// TIA Portal project "Siemens_B3" (V16)

(* hardware
DEVICE "S7-1200 station_1"  S7-1200 Station
   slot 0: "Rack_0"  S7-1200 Rack  Rack  V1.0
   slot 1: "PLC_1"  CPU 1214C DC/DC/DC  6ES7 214-1AG40-0XB0  V4.0
   slot 3: "AQ 1x12BIT_1"  AQ1 signal board  6ES7 232-4HA30-0XB0  V1.0
DEVICE "PC-System_2"  SIMATIC PC station
   slot 0: "SIMATIC PC station"  Rail  SIMATIC PC-Station  V1.0
      slot 125: "Stationmanager"  Station_Manager  V6.0.4
   slot 1: "HMI_RT_2"  WinCC RT Professional  6AV2 105-0xxxx-xxxx  16.0.0.0
   slot 2: "IE general_1"  IE General  IE_CP  V8.2.0
DEVICE "PC-System_1"  SIMATIC PC station
   slot 0: "SIMATIC PC station"  Rail  SIMATIC PC-Station  V1.0
      slot 125: "Stationmanager"  Station_Manager  V6.0.4
   slot 1: "HMI_RT_1"  WinCC RT Advanced  6AV2 104-0xxxx-xxxx  16.0.0.0
      slot 33792: "Computer interface"  Host interface
   slot 2: "IE general_1"  IE General  IE_CP  V8.2.0
*)

// ===== PLC "PLC_1"  CPU 1214C DC/DC/DC =====

VAR_GLOBAL   // PLC tag table "Default tag table"
   "Start" AT %I0.4 : Bool;
   "Emergency" AT %I0.6 : Bool;
   "Stop" AT %I0.5 : Bool;
   "Tag_4" AT %M0.3 : Bool;
   "Move_DL" AT %M0.6 : Bool;
   "On_Timer" AT %M0.7 : Bool;
   "Out_Timer" AT %M1.0 : Bool;
   "Tag_1" AT %Q0.0 : Bool;
   "Tag_2" AT %M3.0 : Bool;
   "Tag_3" AT %M3.1 : Bool;
   "Tag_5" AT %M3.2 : Bool;
   "Tag_6" AT %M3.3 : Bool;
END_VAR

VAR_GLOBAL   // PLC tag table "DI"
   "CB_can_Tank_khuay" AT %I0.0 : Bool;
   "CB_can_Tank_TP" AT %I0.1 : Bool;
   "CB_day_Tank_TP" AT %I0.2 : Bool;
   "CB_loi_BT" AT %I0.3 : Bool;
END_VAR

VAR_GLOBAL   // PLC tag table "AI"
   "CB_can_nang" AT %IW64 : Int;
   "Thoi_gian_Tank_khuay" AT %MD2 : Time;
   "Thoi_gian_khuay" AT %MD4 : Time;
END_VAR

VAR_GLOBAL   // PLC tag table "AQ"
   "Tan_so_BT" AT %QW80 : Int;
END_VAR

VAR_GLOBAL   // PLC tag table "DQ"
   "Van_PV1_1" AT %Q0.1 : Bool;
   "Van_PV1_2" AT %Q0.2 : Bool;
   "Van_PV1_3" AT %Q0.3 : Bool;
   "Van_PV1_4" AT %Q0.4 : Bool;
   "Van_PV1_5" AT %Q0.5 : Bool;
   "Van_PV1_6" AT %Q0.6 : Bool;
   "Dong_co_M1_1" AT %Q0.7 : Bool;
   "Bom_MV1_1" AT %Q1.0 : Bool;
END_VAR

TYPE "UDT_Van"
   STRUCT
      Auto_Man : Bool;
      Start_M : Bool;
      Stop_M : Bool;
      Start_A : Bool;
      Stop_A : Bool;
      Khoi_luong_ban_dau : Real;
      Khoi_luong_nhap_vao : Real;
      Khoi_luong_tong_so_sanh : Real;
      Dieu_kien_OFF : Bool;
      Dieu_kien_ON : Bool;
      Thoi_gian_nhap_vao_khuay : Time;
      Thoi_gian_nhap_vao_rua_CIP : Time;
      Toc_do_nhap_vao : Time;
   END_STRUCT;
END_TYPE

DATA_BLOCK "DB_Analog"   // DB1
{ S7_Optimized_Access := 'TRUE' }
VERSION : 0.1
   VAR
      AI_trung_gian : Real;
      Khoi_luong_tank_khuay : Real;
      Tan_so_INPUT_BT : Real;
      AQ_trung_gian : Real;
   END_VAR
BEGIN
END_DATA_BLOCK

DATA_BLOCK "DB_Van"   // DB2
{ S7_Optimized_Access := 'TRUE' }
VERSION : 0.1
   VAR
      Van_1 : "UDT_Van";
      Van_2 : "UDT_Van";
      Van_3 : "UDT_Van";
      Van_4 : "UDT_Van";
      Van_5 : "UDT_Van";
      Van_6 : "UDT_Van";
   END_VAR
BEGIN
END_DATA_BLOCK

DATA_BLOCK "DB_Tank_khuay"   // DB3
{ S7_Optimized_Access := 'TRUE' }
VERSION : 0.1
   VAR
      Tank_khuay : "UDT_Van";
   END_VAR
BEGIN
END_DATA_BLOCK

DATA_BLOCK "DB_Bom_TP"   // DB4
{ S7_Optimized_Access := 'TRUE' }
VERSION : 0.1
   VAR
      Bom_TP : "UDT_Van";
   END_VAR
BEGIN
END_DATA_BLOCK

// folder: System blocks/Program resources

DATA_BLOCK "Timer_Van_2"   // DB5
{ S7_Optimized_Access := 'TRUE' }
AUTHOR : Simatic
FAMILY : IEC
NAME : IEC_TMR
VERSION : 1.0
// stored: InstanceOfName IEC_TIMER
"IEC_TIMER"
BEGIN
END_DATA_BLOCK

DATA_BLOCK "Timer_Van_1"   // DB6
{ S7_Optimized_Access := 'TRUE' }
AUTHOR : Simatic
FAMILY : IEC
NAME : IEC_TMR
VERSION : 1.0
// stored: InstanceOfName IEC_TIMER
"IEC_TIMER"
BEGIN
END_DATA_BLOCK

DATA_BLOCK "Timer_Tank_khuay"   // DB7
{ S7_Optimized_Access := 'TRUE' }
AUTHOR : Simatic
FAMILY : IEC
NAME : IEC_TMR
VERSION : 1.0
// stored: InstanceOfName IEC_TIMER
"IEC_TIMER"
BEGIN
END_DATA_BLOCK

// folder: (top level)

FUNCTION "FC_Analog" : Void   // FC1, LAD
{ S7_Optimized_Access := 'TRUE' }
VERSION : 0.1
BEGIN

REGION Network 1: ANALOG INPUT cân nặng nước
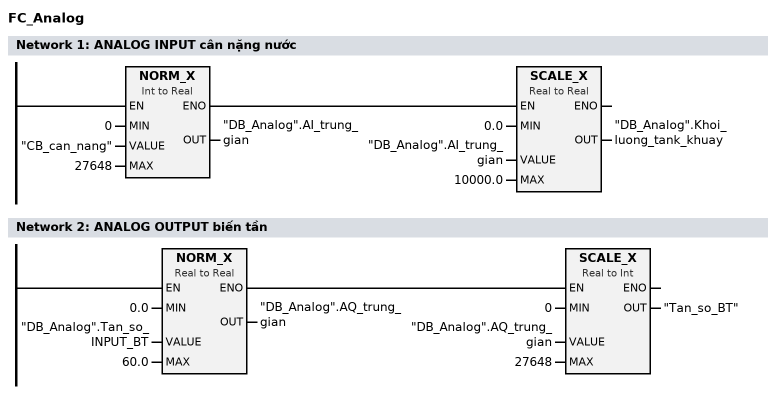
   RUNG wire#powerrail
      { S7_Templates := "[SrcType := Int, DestType := Real]" } Normalize(min := 0, value := "CB_can_nang", max := 27648, out => "DB_Analog".AI_trung_gian)
      { S7_Templates := "[SrcType := Real, DestType := Real]" } Scale(min := 0.0, value := "DB_Analog".AI_trung_gian, max := 10000.0, out => "DB_Analog".Khoi_luong_tank_khuay)
   END_RUNG
   // the same network as SCL:
   "DB_Analog".AI_trung_gian := NORM_X(MIN := 0, VALUE := "CB_can_nang", MAX := 27648);
   "DB_Analog".Khoi_luong_tank_khuay := SCALE_X(MIN := 0.0, VALUE := "DB_Analog".AI_trung_gian, MAX := 10000.0);
END_REGION

REGION Network 2: ANALOG OUTPUT biến tần
   RUNG wire#powerrail
      { S7_Templates := "[SrcType := Real, DestType := Real]" } Normalize(min := 0.0, value := "DB_Analog".Tan_so_INPUT_BT, max := 60.0, out => "DB_Analog".AQ_trung_gian)
      { S7_Templates := "[SrcType := Real, DestType := Int]" } Scale(min := 0, value := "DB_Analog".AQ_trung_gian, max := 27648, out => "Tan_so_BT")
   END_RUNG
   // the same network as SCL:
   "DB_Analog".AQ_trung_gian := NORM_X(MIN := 0.0, VALUE := "DB_Analog".Tan_so_INPUT_BT, MAX := 60.0);
   "Tan_so_BT" := SCALE_X(MIN := 0, VALUE := "DB_Analog".AQ_trung_gian, MAX := 27648);
END_REGION
END_FUNCTION

FUNCTION "FC_Van" : Void   // FC2, LAD
{ S7_Optimized_Access := 'TRUE' }
VERSION : 0.1
   VAR_TEMP   // added for the SCL form of the ladder/FBD networks
      _w1 : Bool;
   END_VAR
BEGIN

REGION Network 1: Van 1: CIP Tank khuấy
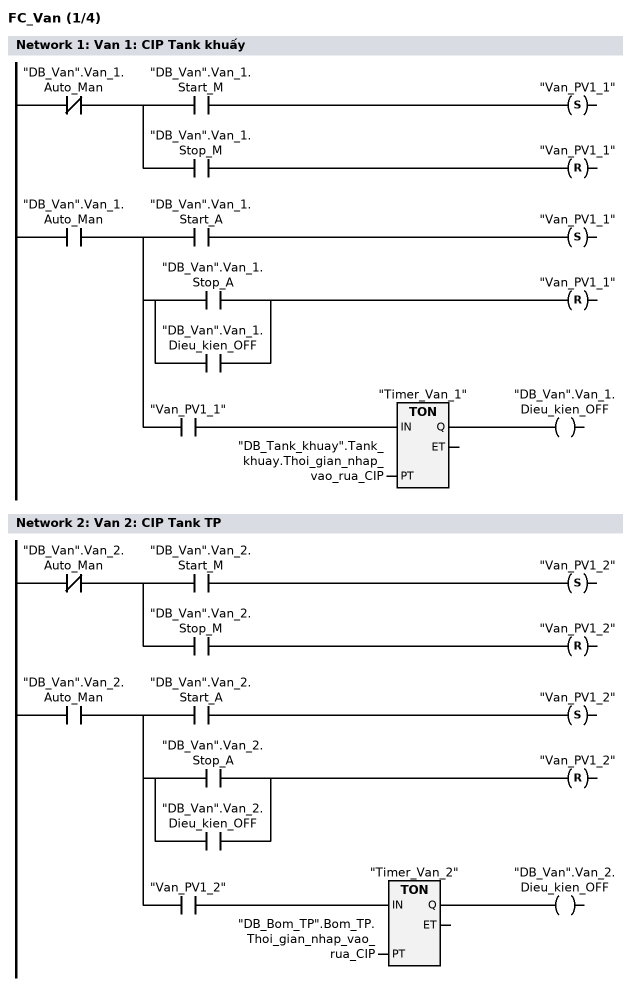
   #_w1 := NOT "DB_Van".Van_1.Auto_Man;
   IF #_w1 AND "DB_Van".Van_1.Start_M THEN "Van_PV1_1" := TRUE; END_IF;
   IF #_w1 AND "DB_Van".Van_1.Stop_M THEN "Van_PV1_1" := FALSE; END_IF;
   IF "DB_Van".Van_1.Auto_Man AND "DB_Van".Van_1.Start_A THEN "Van_PV1_1" := TRUE; END_IF;
   IF "DB_Van".Van_1.Auto_Man AND ("DB_Van".Van_1.Stop_A OR "DB_Van".Van_1.Dieu_kien_OFF) THEN
       "Van_PV1_1" := FALSE;
   END_IF;
   "Timer_Van_1".TON(IN := "DB_Van".Van_1.Auto_Man AND "Van_PV1_1",
                     PT := "DB_Tank_khuay".Tank_khuay.Thoi_gian_nhap_vao_rua_CIP);
   "DB_Van".Van_1.Dieu_kien_OFF := "Timer_Van_1".Q;
END_REGION

REGION Network 2: Van 2: CIP Tank TP
   #_w1 := NOT "DB_Van".Van_2.Auto_Man;
   IF #_w1 AND "DB_Van".Van_2.Start_M THEN "Van_PV1_2" := TRUE; END_IF;
   IF #_w1 AND "DB_Van".Van_2.Stop_M THEN "Van_PV1_2" := FALSE; END_IF;
   IF "DB_Van".Van_2.Auto_Man AND "DB_Van".Van_2.Start_A THEN "Van_PV1_2" := TRUE; END_IF;
   IF "DB_Van".Van_2.Auto_Man AND ("DB_Van".Van_2.Stop_A OR "DB_Van".Van_2.Dieu_kien_OFF) THEN
       "Van_PV1_2" := FALSE;
   END_IF;
   "Timer_Van_2".TON(IN := "DB_Van".Van_2.Auto_Man AND "Van_PV1_2",
                     PT := "DB_Bom_TP".Bom_TP.Thoi_gian_nhap_vao_rua_CIP);
   "DB_Van".Van_2.Dieu_kien_OFF := "Timer_Van_2".Q;
END_REGION

REGION Network 3: Van 3
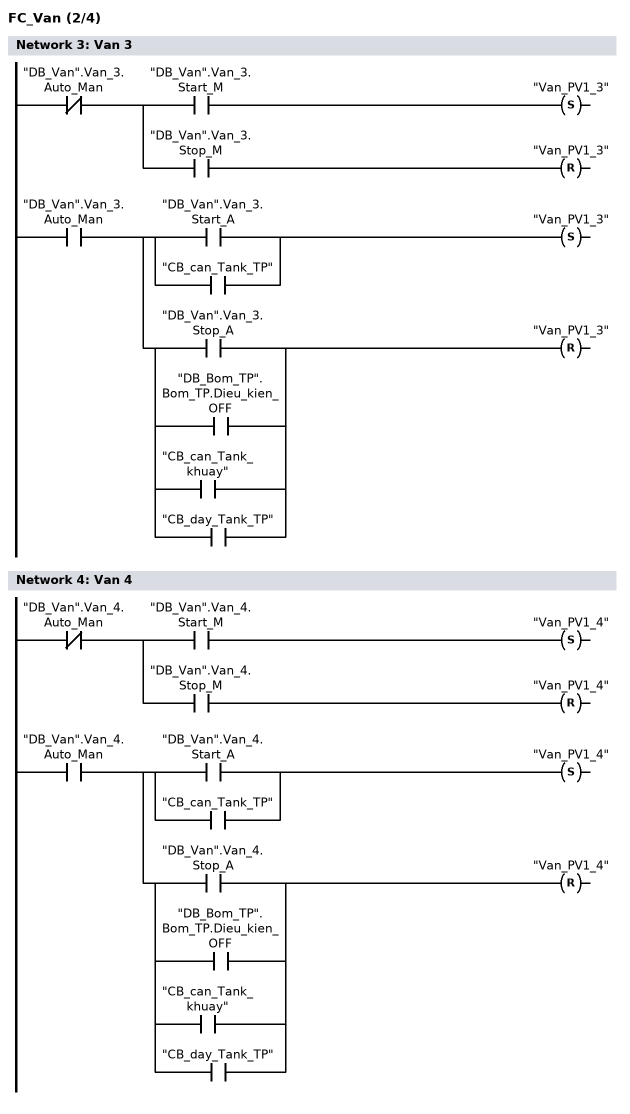
   RUNG wire#powerrail
      I_Contact( "DB_Van".Van_3.Auto_Man )
      wire#w1
      Contact( "DB_Van".Van_3.Start_M )
      S_Coil( "Van_PV1_3" )
   END_RUNG
   RUNG wire#w1
      Contact( "DB_Van".Van_3.Stop_M )
      R_Coil( "Van_PV1_3" )
   END_RUNG
   RUNG wire#powerrail
      Contact( "DB_Van".Van_3.Auto_Man )
      wire#w2
      Contact( "DB_Van".Van_3.Start_A )
      wire#w3
      S_Coil( "Van_PV1_3" )
   END_RUNG
   RUNG wire#w2
      Contact( "CB_can_Tank_TP" )
   END_RUNG wire#w3
   RUNG wire#w2
      Contact( "DB_Van".Van_3.Stop_A )
      wire#w4
      R_Coil( "Van_PV1_3" )
   END_RUNG
   RUNG wire#w2
      Contact( "DB_Bom_TP".Bom_TP.Dieu_kien_OFF )
   END_RUNG wire#w4
   RUNG wire#w2
      Contact( "CB_can_Tank_khuay" )
   END_RUNG wire#w4
   RUNG wire#w2
      Contact( "CB_day_Tank_TP" )
   END_RUNG wire#w4
   // the same network as SCL:
   #_w1 := NOT "DB_Van".Van_3.Auto_Man;
   IF #_w1 AND "DB_Van".Van_3.Start_M THEN "Van_PV1_3" := TRUE; END_IF;
   IF #_w1 AND "DB_Van".Van_3.Stop_M THEN "Van_PV1_3" := FALSE; END_IF;
   IF "DB_Van".Van_3.Auto_Man AND ("DB_Van".Van_3.Start_A OR "CB_can_Tank_TP") THEN
       "Van_PV1_3" := TRUE;
   END_IF;
   IF "DB_Van".Van_3.Auto_Man AND ("DB_Van".Van_3.Stop_A OR "DB_Bom_TP".Bom_TP.Dieu_kien_OFF OR "CB_can_Tank_khuay" OR "CB_day_Tank_TP") THEN
       "Van_PV1_3" := FALSE;
   END_IF;
END_REGION

REGION Network 4: Van 4
   RUNG wire#powerrail
      I_Contact( "DB_Van".Van_4.Auto_Man )
      wire#w1
      Contact( "DB_Van".Van_4.Start_M )
      S_Coil( "Van_PV1_4" )
   END_RUNG
   RUNG wire#w1
      Contact( "DB_Van".Van_4.Stop_M )
      R_Coil( "Van_PV1_4" )
   END_RUNG
   RUNG wire#powerrail
      Contact( "DB_Van".Van_4.Auto_Man )
      wire#w2
      Contact( "DB_Van".Van_4.Start_A )
      wire#w3
      S_Coil( "Van_PV1_4" )
   END_RUNG
   RUNG wire#w2
      Contact( "CB_can_Tank_TP" )
   END_RUNG wire#w3
   RUNG wire#w2
      Contact( "DB_Van".Van_4.Stop_A )
      wire#w4
      R_Coil( "Van_PV1_4" )
   END_RUNG
   RUNG wire#w2
      Contact( "DB_Bom_TP".Bom_TP.Dieu_kien_OFF )
   END_RUNG wire#w4
   RUNG wire#w2
      Contact( "CB_can_Tank_khuay" )
   END_RUNG wire#w4
   RUNG wire#w2
      Contact( "CB_day_Tank_TP" )
   END_RUNG wire#w4
   // the same network as SCL:
   #_w1 := NOT "DB_Van".Van_4.Auto_Man;
   IF #_w1 AND "DB_Van".Van_4.Start_M THEN "Van_PV1_4" := TRUE; END_IF;
   IF #_w1 AND "DB_Van".Van_4.Stop_M THEN "Van_PV1_4" := FALSE; END_IF;
   IF "DB_Van".Van_4.Auto_Man AND ("DB_Van".Van_4.Start_A OR "CB_can_Tank_TP") THEN
       "Van_PV1_4" := TRUE;
   END_IF;
   IF "DB_Van".Van_4.Auto_Man AND ("DB_Van".Van_4.Stop_A OR "DB_Bom_TP".Bom_TP.Dieu_kien_OFF OR "CB_can_Tank_khuay" OR "CB_day_Tank_TP") THEN
       "Van_PV1_4" := FALSE;
   END_IF;
END_REGION

REGION Network 5: Van 5 - Cấp nước
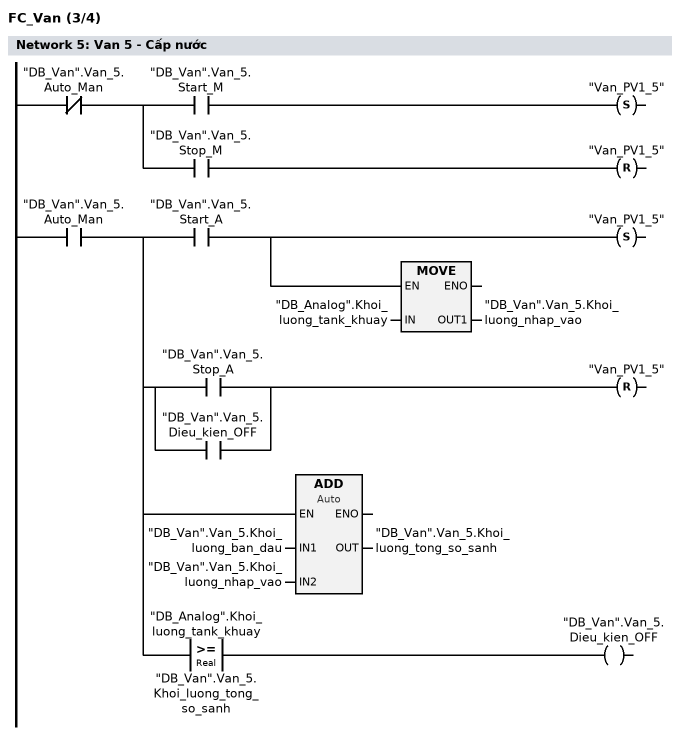
   RUNG wire#powerrail
      I_Contact( "DB_Van".Van_5.Auto_Man )
      wire#w1
      Contact( "DB_Van".Van_5.Start_M )
      S_Coil( "Van_PV1_5" )
   END_RUNG
   RUNG wire#w1
      Contact( "DB_Van".Van_5.Stop_M )
      R_Coil( "Van_PV1_5" )
   END_RUNG
   RUNG wire#powerrail
      Contact( "DB_Van".Van_5.Auto_Man )
      wire#w2
      Contact( "DB_Van".Van_5.Start_A )
      wire#w3
      S_Coil( "Van_PV1_5" )
   END_RUNG
   RUNG wire#w3
      Move(in := "DB_Analog".Khoi_luong_tank_khuay, out1 => "DB_Van".Van_5.Khoi_luong_nhap_vao)
   END_RUNG
   RUNG wire#w2
      Contact( "DB_Van".Van_5.Stop_A )
      wire#w4
      R_Coil( "Van_PV1_5" )
   END_RUNG
   RUNG wire#w2
      Contact( "DB_Van".Van_5.Dieu_kien_OFF )
   END_RUNG wire#w4
   RUNG wire#w2
      Add(in1 := "DB_Van".Van_5.Khoi_luong_ban_dau, in2 := "DB_Van".Van_5.Khoi_luong_nhap_vao, out => "DB_Van".Van_5.Khoi_luong_tong_so_sanh)
   END_RUNG
   RUNG wire#w2
      { S7_Templates := "SrcType := Real" } GE_Contact(in1 := "DB_Analog".Khoi_luong_tank_khuay, in2 := "DB_Van".Van_5.Khoi_luong_tong_so_sanh)
      Coil( "DB_Van".Van_5.Dieu_kien_OFF )
   END_RUNG
   // the same network as SCL:
   #_w1 := NOT "DB_Van".Van_5.Auto_Man;
   IF #_w1 AND "DB_Van".Van_5.Start_M THEN "Van_PV1_5" := TRUE; END_IF;
   IF #_w1 AND "DB_Van".Van_5.Stop_M THEN "Van_PV1_5" := FALSE; END_IF;
   IF "DB_Van".Van_5.Auto_Man AND "DB_Van".Van_5.Start_A THEN
       "Van_PV1_5" := TRUE;
       "DB_Van".Van_5.Khoi_luong_nhap_vao := "DB_Analog".Khoi_luong_tank_khuay;
   END_IF;
   IF "DB_Van".Van_5.Auto_Man AND ("DB_Van".Van_5.Stop_A OR "DB_Van".Van_5.Dieu_kien_OFF) THEN
       "Van_PV1_5" := FALSE;
   END_IF;
   IF "DB_Van".Van_5.Auto_Man THEN
       "DB_Van".Van_5.Khoi_luong_tong_so_sanh := "DB_Van".Van_5.Khoi_luong_ban_dau + "DB_Van".Van_5.Khoi_luong_nhap_vao;
   END_IF;
   "DB_Van".Van_5.Dieu_kien_OFF := "DB_Van".Van_5.Auto_Man AND ("DB_Analog".Khoi_luong_tank_khuay >= "DB_Van".Van_5.Khoi_luong_tong_so_sanh);
END_REGION

REGION Network 6: Van 6 - Cấp cồn
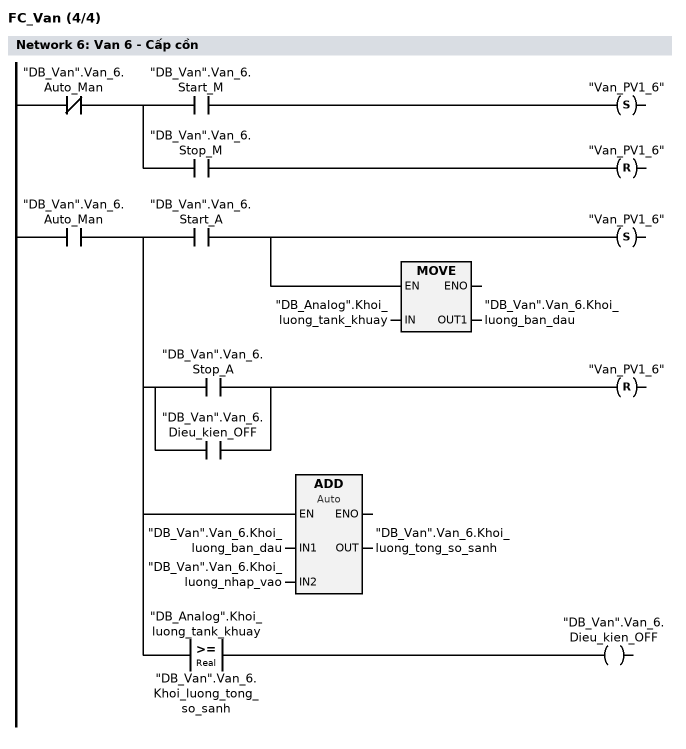
   RUNG wire#powerrail
      I_Contact( "DB_Van".Van_6.Auto_Man )
      wire#w1
      Contact( "DB_Van".Van_6.Start_M )
      S_Coil( "Van_PV1_6" )
   END_RUNG
   RUNG wire#w1
      Contact( "DB_Van".Van_6.Stop_M )
      R_Coil( "Van_PV1_6" )
   END_RUNG
   RUNG wire#powerrail
      Contact( "DB_Van".Van_6.Auto_Man )
      wire#w2
      Contact( "DB_Van".Van_6.Start_A )
      wire#w3
      S_Coil( "Van_PV1_6" )
   END_RUNG
   RUNG wire#w3
      Move(in := "DB_Analog".Khoi_luong_tank_khuay, out1 => "DB_Van".Van_6.Khoi_luong_ban_dau)
   END_RUNG
   RUNG wire#w2
      Contact( "DB_Van".Van_6.Stop_A )
      wire#w4
      R_Coil( "Van_PV1_6" )
   END_RUNG
   RUNG wire#w2
      Contact( "DB_Van".Van_6.Dieu_kien_OFF )
   END_RUNG wire#w4
   RUNG wire#w2
      Add(in1 := "DB_Van".Van_6.Khoi_luong_ban_dau, in2 := "DB_Van".Van_6.Khoi_luong_nhap_vao, out => "DB_Van".Van_6.Khoi_luong_tong_so_sanh)
   END_RUNG
   RUNG wire#w2
      { S7_Templates := "SrcType := Real" } GE_Contact(in1 := "DB_Analog".Khoi_luong_tank_khuay, in2 := "DB_Van".Van_6.Khoi_luong_tong_so_sanh)
      Coil( "DB_Van".Van_6.Dieu_kien_OFF )
   END_RUNG
   // the same network as SCL:
   #_w1 := NOT "DB_Van".Van_6.Auto_Man;
   IF #_w1 AND "DB_Van".Van_6.Start_M THEN "Van_PV1_6" := TRUE; END_IF;
   IF #_w1 AND "DB_Van".Van_6.Stop_M THEN "Van_PV1_6" := FALSE; END_IF;
   IF "DB_Van".Van_6.Auto_Man AND "DB_Van".Van_6.Start_A THEN
       "Van_PV1_6" := TRUE;
       "DB_Van".Van_6.Khoi_luong_ban_dau := "DB_Analog".Khoi_luong_tank_khuay;
   END_IF;
   IF "DB_Van".Van_6.Auto_Man AND ("DB_Van".Van_6.Stop_A OR "DB_Van".Van_6.Dieu_kien_OFF) THEN
       "Van_PV1_6" := FALSE;
   END_IF;
   IF "DB_Van".Van_6.Auto_Man THEN
       "DB_Van".Van_6.Khoi_luong_tong_so_sanh := "DB_Van".Van_6.Khoi_luong_ban_dau + "DB_Van".Van_6.Khoi_luong_nhap_vao;
   END_IF;
   "DB_Van".Van_6.Dieu_kien_OFF := "DB_Van".Van_6.Auto_Man AND ("DB_Analog".Khoi_luong_tank_khuay >= "DB_Van".Van_6.Khoi_luong_tong_so_sanh);
END_REGION
END_FUNCTION

FUNCTION "FC_Tank_khuay" : Void   // FC3, LAD
{ S7_Optimized_Access := 'TRUE' }
VERSION : 0.1
   VAR_TEMP   // added for the SCL form of the ladder/FBD networks
      _w1 : Bool;
      _w2 : Bool;
   END_VAR
BEGIN

REGION Network 1: Động cơ M1.1 - Biến tần, Timer
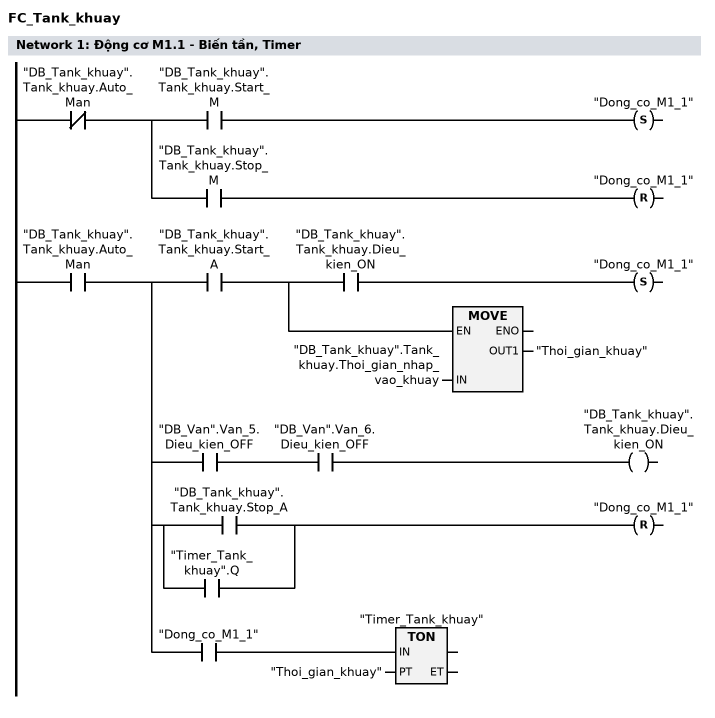
   #_w1 := NOT "DB_Tank_khuay".Tank_khuay.Auto_Man;
   IF #_w1 AND "DB_Tank_khuay".Tank_khuay.Start_M THEN "Dong_co_M1_1" := TRUE; END_IF;
   IF #_w1 AND "DB_Tank_khuay".Tank_khuay.Stop_M THEN "Dong_co_M1_1" := FALSE; END_IF;
   #_w2 := "DB_Tank_khuay".Tank_khuay.Auto_Man AND "DB_Tank_khuay".Tank_khuay.Start_A;
   IF #_w2 AND "DB_Tank_khuay".Tank_khuay.Dieu_kien_ON THEN "Dong_co_M1_1" := TRUE; END_IF;
   IF #_w2 THEN "Thoi_gian_khuay" := "DB_Tank_khuay".Tank_khuay.Thoi_gian_nhap_vao_khuay; END_IF;
   "DB_Tank_khuay".Tank_khuay.Dieu_kien_ON := "DB_Tank_khuay".Tank_khuay.Auto_Man AND "DB_Van".Van_5.Dieu_kien_OFF AND "DB_Van".Van_6.Dieu_kien_OFF;
   IF "DB_Tank_khuay".Tank_khuay.Auto_Man AND ("DB_Tank_khuay".Tank_khuay.Stop_A OR "Timer_Tank_khuay".Q) THEN
       "Dong_co_M1_1" := FALSE;
   END_IF;
   "Timer_Tank_khuay".TON(IN := "DB_Tank_khuay".Tank_khuay.Auto_Man AND "Dong_co_M1_1", PT := "Thoi_gian_khuay");
END_REGION
END_FUNCTION

FUNCTION "FC_Bom_TP" : Void   // FC4, LAD
{ S7_Optimized_Access := 'TRUE' }
VERSION : 0.1
   VAR_TEMP   // added for the SCL form of the ladder/FBD networks
      _w1 : Bool;
   END_VAR
BEGIN

REGION Network 1: Bơm thành phẩm
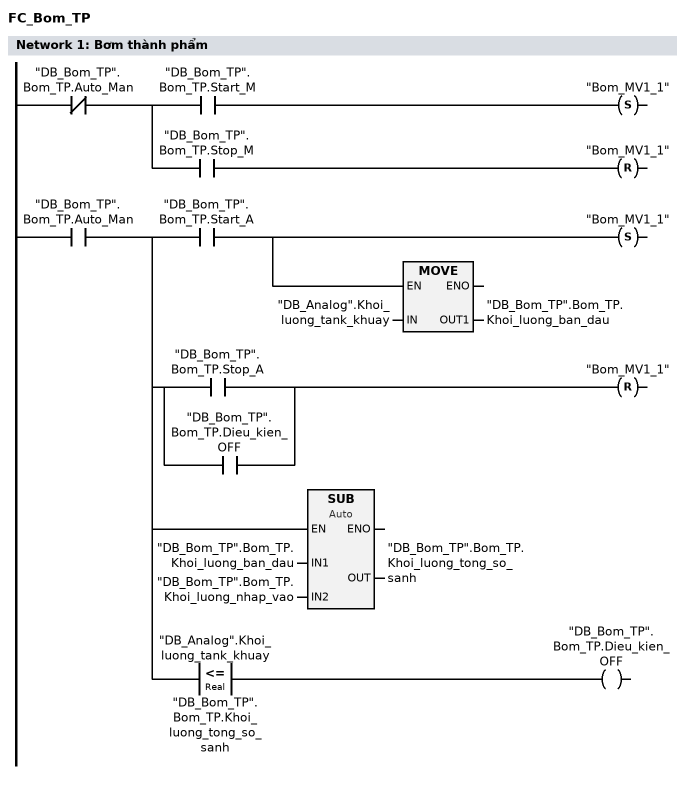
   RUNG wire#powerrail
      I_Contact( "DB_Bom_TP".Bom_TP.Auto_Man )
      wire#w1
      Contact( "DB_Bom_TP".Bom_TP.Start_M )
      S_Coil( "Bom_MV1_1" )
   END_RUNG
   RUNG wire#w1
      Contact( "DB_Bom_TP".Bom_TP.Stop_M )
      R_Coil( "Bom_MV1_1" )
   END_RUNG
   RUNG wire#powerrail
      Contact( "DB_Bom_TP".Bom_TP.Auto_Man )
      wire#w2
      Contact( "DB_Bom_TP".Bom_TP.Start_A )
      wire#w3
      S_Coil( "Bom_MV1_1" )
   END_RUNG
   RUNG wire#w3
      Move(in := "DB_Analog".Khoi_luong_tank_khuay, out1 => "DB_Bom_TP".Bom_TP.Khoi_luong_ban_dau)
   END_RUNG
   RUNG wire#w2
      Contact( "DB_Bom_TP".Bom_TP.Stop_A )
      wire#w4
      R_Coil( "Bom_MV1_1" )
   END_RUNG
   RUNG wire#w2
      Contact( "DB_Bom_TP".Bom_TP.Dieu_kien_OFF )
   END_RUNG wire#w4
   RUNG wire#w2
      Sub(in1 := "DB_Bom_TP".Bom_TP.Khoi_luong_ban_dau, in2 := "DB_Bom_TP".Bom_TP.Khoi_luong_nhap_vao, out => "DB_Bom_TP".Bom_TP.Khoi_luong_tong_so_sanh)
   END_RUNG
   RUNG wire#w2
      { S7_Templates := "SrcType := Real" } LE_Contact(in1 := "DB_Analog".Khoi_luong_tank_khuay, in2 := "DB_Bom_TP".Bom_TP.Khoi_luong_tong_so_sanh)
      Coil( "DB_Bom_TP".Bom_TP.Dieu_kien_OFF )
   END_RUNG
   // the same network as SCL:
   #_w1 := NOT "DB_Bom_TP".Bom_TP.Auto_Man;
   IF #_w1 AND "DB_Bom_TP".Bom_TP.Start_M THEN "Bom_MV1_1" := TRUE; END_IF;
   IF #_w1 AND "DB_Bom_TP".Bom_TP.Stop_M THEN "Bom_MV1_1" := FALSE; END_IF;
   IF "DB_Bom_TP".Bom_TP.Auto_Man AND "DB_Bom_TP".Bom_TP.Start_A THEN
       "Bom_MV1_1" := TRUE;
       "DB_Bom_TP".Bom_TP.Khoi_luong_ban_dau := "DB_Analog".Khoi_luong_tank_khuay;
   END_IF;
   IF "DB_Bom_TP".Bom_TP.Auto_Man AND ("DB_Bom_TP".Bom_TP.Stop_A OR "DB_Bom_TP".Bom_TP.Dieu_kien_OFF) THEN
       "Bom_MV1_1" := FALSE;
   END_IF;
   IF "DB_Bom_TP".Bom_TP.Auto_Man THEN
       "DB_Bom_TP".Bom_TP.Khoi_luong_tong_so_sanh := "DB_Bom_TP".Bom_TP.Khoi_luong_ban_dau - "DB_Bom_TP".Bom_TP.Khoi_luong_nhap_vao;
   END_IF;
   "DB_Bom_TP".Bom_TP.Dieu_kien_OFF := "DB_Bom_TP".Bom_TP.Auto_Man AND ("DB_Analog".Khoi_luong_tank_khuay <= "DB_Bom_TP".Bom_TP.Khoi_luong_tong_so_sanh);
END_REGION
END_FUNCTION

ORGANIZATION_BLOCK "Main"   // OB1, LAD, ProgramCycle
TITLE = "Main Program Sweep (Cycle)"
{ S7_Optimized_Access := 'TRUE' }
VERSION : 0.1
   VAR_INPUT
      Initial_Call : Bool;   // Initial call of this OB
      Remanence : Bool;   // =True, if remanent data are available
   END_VAR
BEGIN

REGION Network 1
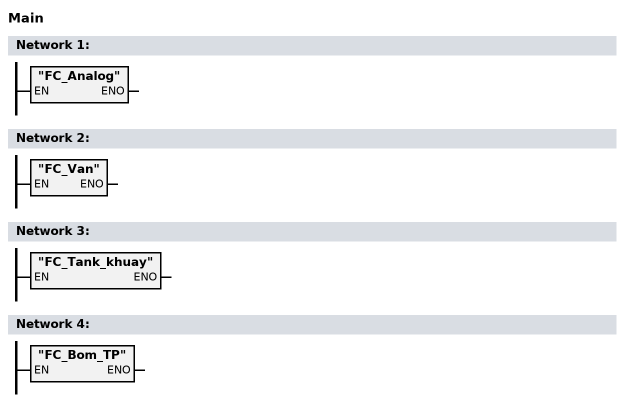
   RUNG wire#powerrail
      "FC_Analog"()
   END_RUNG
   // the same network as SCL:
   "FC_Analog"();
END_REGION

REGION Network 2
   RUNG wire#powerrail
      "FC_Van"()
   END_RUNG
   // the same network as SCL:
   "FC_Van"();
END_REGION

REGION Network 3
   RUNG wire#powerrail
      "FC_Tank_khuay"()
   END_RUNG
   // the same network as SCL:
   "FC_Tank_khuay"();
END_REGION

REGION Network 4
   RUNG wire#powerrail
      "FC_Bom_TP"()
   END_RUNG
   // the same network as SCL:
   "FC_Bom_TP"();
END_REGION
END_ORGANIZATION_BLOCK

(* ===== HMI "HMI_RT_2" =====
system functions are stored by id; their names below are inferred from use
connection "HMI_Connection_1": S71200_TCP_IP, SCADA_S7_1200

HMI tags "DI"
   "CB_can_Tank_khuay" : Bool = PLC CB_can_Tank_khuay AT %I0.0, 500 ms
   "CB_can_Tank_TP" : Bool = PLC CB_can_Tank_TP AT %I0.1, 500 ms
   "CB_day_Tank_TP" : Bool = PLC CB_day_Tank_TP AT %I0.2, 500 ms
   "CB_loi_BT" : Bool = PLC CB_loi_BT AT %I0.3, 500 ms

HMI tags "DQ"
   "Van_PV1_1" : Bool = PLC Van_PV1_1 AT %Q0.1, 500 ms
   "Van_PV1_2" : Bool = PLC Van_PV1_2 AT %Q0.2, 500 ms
   "Van_PV1_3" : Bool = PLC Van_PV1_3 AT %Q0.3, 500 ms
   "Van_PV1_4" : Bool = PLC Van_PV1_4 AT %Q0.4, 500 ms
   "Van_PV1_5" : Bool = PLC Van_PV1_5 AT %Q0.5, 500 ms
   "Van_PV1_6" : Bool = PLC Van_PV1_6 AT %Q0.6, 500 ms
   "Dong_co_M1_1" : Bool = PLC Dong_co_M1_1 AT %Q0.7, 500 ms
   "Bom_MV1_1" : Bool = PLC Bom_MV1_1 AT %Q1.0, 500 ms

HMI tags "AI"
   "CB_can_nang" : Int = PLC CB_can_nang AT %IW64, 500 ms

HMI tags "AQ"
   "Tan_so_BT" : Int = PLC Tan_so_BT AT %QW80, 500 ms

HMI tags "Van"
   "DB_Van_Van_1" : UDT_Van = PLC DB_Van.Van_1, 500 ms
   "DB_Van_Van_2" : UDT_Van = PLC DB_Van.Van_2, 500 ms
   "DB_Van_Van_3" : UDT_Van = PLC DB_Van.Van_3, 500 ms
   "DB_Van_Van_4" : UDT_Van = PLC DB_Van.Van_4, 500 ms
   "DB_Van_Van_5" : UDT_Van = PLC DB_Van.Van_5, 500 ms
   "DB_Van_Van_6" : UDT_Van = PLC DB_Van.Van_6, 500 ms

HMI tags "Bom_TP"
   "DB_Bom_TP_Bom_TP" : UDT_Van = PLC DB_Bom_TP.Bom_TP, 500 ms

HMI tags "Tank_khuay"
   "DB_Tank_khuay_Tank_khuay" : UDT_Van = PLC DB_Tank_khuay.Tank_khuay, 500 ms

HMI tags "Analog"
   "DB_Analog_AI_trung_gian" : Real = PLC DB_Analog.AI_trung_gian, 500 ms
   "DB_Analog_Khoi_luong_tank_khuay" : Real = PLC DB_Analog.Khoi_luong_tank_khuay, 500 ms
   "DB_Analog_Tan_so_INPUT_BT" : Real = PLC DB_Analog.Tan_so_INPUT_BT, 500 ms
   "DB_Analog_AQ_trung_gian" : Real = PLC DB_Analog.AQ_trung_gian, 500 ms

screen "SC_Main" 1920x1080
   TextField "Text field_1" at 874,23 size 173x25; Text 'Hệ thống pha trộn'
   Clock "Clock_1" at 1573,11 size 120x68
   GraphicView "Graphic view_1" at 0,0 size 70x69; Picture "Graphic_1"
   TextField "Text field_2" at 554,585 size 135x19; Text 'BẢNG ĐIỀU KHIỂN'
   SymbolLibrary "Symbol library_7" at 580,409 size 73x120
      Appearance <- "Van_PV1_1"
   TextField "Text field_3" at 529,624 size 84x19; Text 'AUTO/MAN'
   TextField "Text field_4" at 530,701 size 79x19; Text 'COMMAND'
   Button "Button_1" at 529,653 size 80x30; TextOff 'MAN'
      on Click: SetBit("Auto_Man")
   Button "Button_2" at 629,654 size 80x30; TextOff 'AUTO'
      on Click: SetBit("Auto_Man")
   Button "Button_3" at 529,728 size 80x30; TextOff 'START'
      on PressLeft: SetBit("Start_M")
      on ReleaseLeft: SetBit("Start_M")
   Button "Button_4" at 629,727 size 80x30; TextOff 'STOP'
      on PressLeft: SetBit("Stop_M")
      on ReleaseLeft: SetBit("Stop_M")

screen "SC_System" 1920x1080
   TextField "Text field_1" at 874,23 size 173x25; Text 'Hệ thống pha trộn'
   Clock "Clock_1" at 1573,11 size 120x68
   GraphicView "Graphic view_1" at 0,0 size 70x69; Picture "Graphic_1"
   SymbolLibrary "Symbol library_7" at 281,261 size 40x56
      Appearance <- "Van_PV1_1"
   SymbolLibrary "Symbol library_1" at 347,506 size 244x324
   SymbolLibrary "Symbol library_2" at 420,403 size 241x322
   SymbolLibrary "Symbol library_3" at 814,892 size 102x84
   SymbolLibrary "Symbol library_4" at 1123,506 size 244x324
   SymbolLibrary "Symbol library_6" at 317,301 size 59x13
   SymbolLibrary "Symbol library_8" at 119,301 size 167x13
   SymbolLibrary "Symbol library_9" at 764,165 size 40x56
      Appearance <- "Van_PV1_1"
   SymbolLibrary "Symbol library_10" at 800,205 size 27x13
   SymbolLibrary "Symbol library_11" at 602,205 size 167x13
   SymbolLibrary "Symbol library_12" at 366,301 size 25x25
   SymbolLibrary "Symbol library_13" at 378,325 size 13x188
   SymbolLibrary "Symbol library_14" at 822,205 size 25x25
   SymbolLibrary "Symbol library_15" at 834,228 size 13x233
*)

(* ===== HMI "HMI_RT_1" =====
system functions are stored by id; their names below are inferred from use
connection "HMI_Connection_3": ETHERNET, S7_1200_OMS

HMI tags "DQ_2"
   "Bom_MV1_1" : Bool = PLC Bom_MV1_1 AT %Q1.0, 500 ms
   "Dong_co_M1_1" : Bool = PLC Dong_co_M1_1 AT %Q0.7, 500 ms
   "Van_PV1_1" : Bool = PLC Van_PV1_1 AT %Q0.1, 500 ms
   "Van_PV1_2" : Bool = PLC Van_PV1_2 AT %Q0.2, 500 ms
   "Van_PV1_3" : Bool = PLC Van_PV1_3 AT %Q0.3, 500 ms
   "Van_PV1_4" : Bool = PLC Van_PV1_4 AT %Q0.4, 500 ms
   "Van_PV1_5" : Bool = PLC Van_PV1_5 AT %Q0.5, 500 ms
   "Van_PV1_6" : Bool = PLC Van_PV1_6 AT %Q0.6, 500 ms

HMI tags "DI_2"
   "CB_can_Tank_khuay" : Bool = PLC CB_can_Tank_khuay AT %I0.0, 1 s
   "CB_can_Tank_TP" : Bool = PLC CB_can_Tank_TP AT %I0.1, 1 s
   "CB_day_Tank_TP" : Bool = PLC CB_day_Tank_TP AT %I0.2, 1 s
   "CB_loi_BT" : Bool = PLC CB_loi_BT AT %I0.3, 1 s

HMI tags "AQ_2"
   "Tan_so_BT" : Int = PLC Tan_so_BT AT %QW80, 1 s

HMI tags "AI_2"
   "CB_can_nang" : Int = PLC CB_can_nang AT %IW64, 1 s

HMI tags "Van_2"
   "DB_Van_Van_1" : UDT_Van = PLC DB_Van.Van_1, 1 s
   "DB_Van_Van_2" : UDT_Van = PLC DB_Van.Van_2, 1 s
   "DB_Van_Van_3" : UDT_Van = PLC DB_Van.Van_3, 1 s
   "DB_Van_Van_4" : UDT_Van = PLC DB_Van.Van_4, 1 s
   "DB_Van_Van_5" : UDT_Van = PLC DB_Van.Van_5, 1 s
   "DB_Van_Van_6" : UDT_Van = PLC DB_Van.Van_6, 1 s

screen "Main" 1920x1080
   TextField "Text field_1" at 874,23 size 173x25; Text 'Hệ thống pha trộn'
   Clock "Clock_1" at 1763,18 size 120x68
   GraphicView "Graphic view_1" at 0,0 size 70x69; Picture "Graphic_1"
   TextField "Text field_2" at 554,585 size 135x19; Text 'BẢNG ĐIỀU KHIỂN'
   SymbolLibrary "Symbol library_7" at 588,415 size 73x120
      Appearance <- "Van_PV1_1"
   TextField "Text field_3" at 529,624 size 84x19; Text 'AUTO/MAN'
   TextField "Text field_4" at 530,701 size 79x19; Text 'COMMAND'
   Button "Button_1" at 529,653 size 80x30; TextOff 'MAN'
      Appearance <- "Auto_Man"
      on Change: SetBit("Auto_Man")
   Button "Button_2" at 629,654 size 80x30; TextOff 'AUTO'
      on Change: SetBit("Auto_Man")
      Appearance <- "Auto_Man"
   Button "Button_3" at 529,728 size 80x30; TextOff 'START'
      on Press: SetBit("Start_M")
      on Release: SetBit("Start_M")
      Appearance <- "Start_M"
   Button "Button_4" at 629,727 size 80x30; TextOff 'STOP'
      on Press: SetBit("Stop_M")
      on Release: SetBit("Stop_M")
      Appearance <- "Stop_M"
*)